DEVICE_TYPE Soft_dPAC (* Synthetic test fixture *)
  PACKAGE SE.DPAC;
END_DEVICE_TYPE
